{attribute addProperty BoxType "AX8620-0000-0029"}
{attribute addProperty Id "Controlword_for_axisAT %I*Controlword_for_axis_FF97049B162"}
{attribute addProperty CRC "1504721345"}
{attribute addProperty SizeInBites "16"}
{attribute addProperty SizeInBytes "2"}
TYPE PSM_Controlword_for_axis_59B039C1 :
STRUCT
	{attribute addProperty Name "Controlword_for_axis"}
	Controlword_for_axis AT %I* : Controlword_for_axis_FF97049B;
END_STRUCT
END_TYPE

(* stored: Version 1.2.0.0, ProductVersion 3.1.4024.9
   DUT PSM_Controlword_for_axis_59B039C1: Id {9eb232f7-08a5-4ebb-9eaf-8992cfdeed58} *)
